(* PLC project Untitled1, Beckhoff Automation GmbH TF6420 Database Server Query Analyser 1.0.0.0 *)
(* stored: creationDateTime 2023-11-08T08:31:45, modificationDateTime 2023-11-08T08:31:45 *)

TYPE ST_Masurdata : STRUCT
  id : LINT;
  time2 : REAL;
  primary_power : REAL;
  secondary_power : REAL;
  phase_shift : REAL;
  frequency : REAL;
  flux_density : REAL;
  Meta_id : LINT;
END_STRUCT;
END_TYPE
